(* Logix 5000 project; controller cal1632 1756-L62 rev 16.20; software revision 16.05; part 52 of 61 *)
(* tags used below, declared in another part *)
   FAULT : BOOL;
   HMI : BOOL;
   p01_param_turret_dia_ft : REAL;
   p01r09_pb_global_reset : BOOL;
   p02_real_from_hmi : hmi_real;
   p29_ai_wa_amps : REAL;
   p29_ai_wa_dia_ft : REAL;
   p29_ai_wa_speed : REAL;
   p29_ai_wa_torque : REAL;
   p29_ai_wb_amps : REAL;
   p29_ai_wb_dia_ft : REAL;
   p29_ai_wb_speed : REAL;
   p29_ai_wb_torque : REAL;
   p29_ai_wdr_dia_in : REAL;
   p29_ai_wdr_lc : REAL;
   p29_ai_wdr_turret_amps : REAL;
   p29_ai_wdr_turret_hz : REAL;
   p29_ai_wdr_turret_speed : REAL;
   p29_ao_wda_vfd : REAL;
   p29_ao_wdb_vfd : REAL;
   p29_ao_wdr_turret_selected_speed : REAL;
   p29_ao_wdra_selected_speed : REAL;
   p29_ao_wdrb_selected_speed : REAL;
   p29_di_wdr_turret : acs800_di_normal;
   p29_dint_to_hmi : DINT[16];
   p29_do_wdr_turret : acs800_do_normal;
   p29_param_wa_gear_ratio : REAL;
   p29_param_wb_gear_ratio : REAL;
   p29_param_wdt_gear_ratio : REAL;
   p29_real_to_hmi : REAL[112];
   p29_wda_control_word : INT;
   p29_wda_status_word : INT;
   p29_wda_vfd_input_max : REAL;
   p29_wda_vfd_input_min : REAL;
   p29_wda_vfd_output_max : REAL;
   p29_wda_vfd_output_min : REAL;
   p29_wdb_control_word : INT;
   p29_wdb_status_word : INT;
   p29_wdb_vfd_input_max : REAL;
   p29_wdb_vfd_input_min : REAL;
   p29_wdb_vfd_output_max : REAL;
   p29_wdb_vfd_output_min : REAL;
   p29r01 : routine;
   p29r03_wa_tq_fifo : CONTROL;
   p29r04 : routine;
   p29r04_timer_fault : TIMER[4];
   p29r04_timer_warning : TIMER[4];
   p29r04_wda_vfd_out_scaling : SYS_SCP;
   p29r04_wdb_vfd_out_scaling : SYS_SCP;
   p29r04_wdr_turret_speed_to_vfd : SYS_SPEED_TO_VFD;
   p29r04_wdra_speed_to_vfd : SYS_SPEED_TO_VFD;
   p29r04_wdrb_speed_to_vfd : SYS_SPEED_TO_VFD;
   p29r05 : routine;
   p29r05_timer_fault : TIMER[4];
   p29r05_timer_warning : TIMER[4];
   p29r06 : routine;
   p29r06_ave_wdr_lc : REAL;
   p29r06_lc_buffer : REAL[20];
   p29r06_sample_timer : TIMER;
   p29r06_timer_fault : TIMER[4];
   p29r06_timer_warning : TIMER[4];
   p29r06_unload : REAL;
   p29r06_wdr_lc_ave_ctrl : CONTROL;
   p29r06_wdr_lc_fifo : CONTROL;
   p29r13_ai_wa_footage_ft : REAL;
   p29r13_ai_wb_footage_ft : REAL;
   p29r15_ao_torque : REAL;
   p29r15_wdra_active : BOOL;
   p29r16_ao_torque : REAL;
   p29r16_wdrb_active : BOOL;
   p29r17_winder_a_avg_diam_inch : REAL;
   p29r18_winder_b_avg_diam_inch : REAL;
   p29r20_index_complete : BOOL;
   turret_in_position : BOOL;   // Turret In Position
(* P29_Winder, continued *)

ROUTINE R04_Output   (* ladder *)
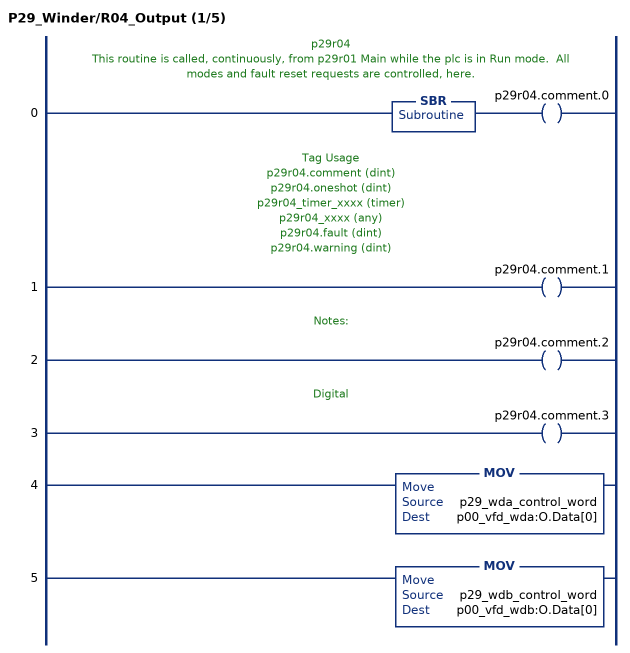
   // p29r04
   // This routine is called, continuously, from p29r01 Main while the plc is in Run mode.  All modes and fault reset requests are controlled, here.
   0: SBR()OTE(p29r04.comment.0);
   // Tag Usage
   // p29r04.comment (dint)
   // p29r04.oneshot (dint)
   // p29r04_timer_xxxx (timer)
   // p29r04_xxxx (any)
   // p29r04.fault (dint)
   // p29r04.warning (dint)
   1: OTE(p29r04.comment.1);
   // Notes:
   2: OTE(p29r04.comment.2);
   // Digital
   3: OTE(p29r04.comment.3);
   4: MOV(p29_wda_control_word,p00_vfd_wda:O.Data[0]);
   5: MOV(p29_wdb_control_word,p00_vfd_wdb:O.Data[0]);
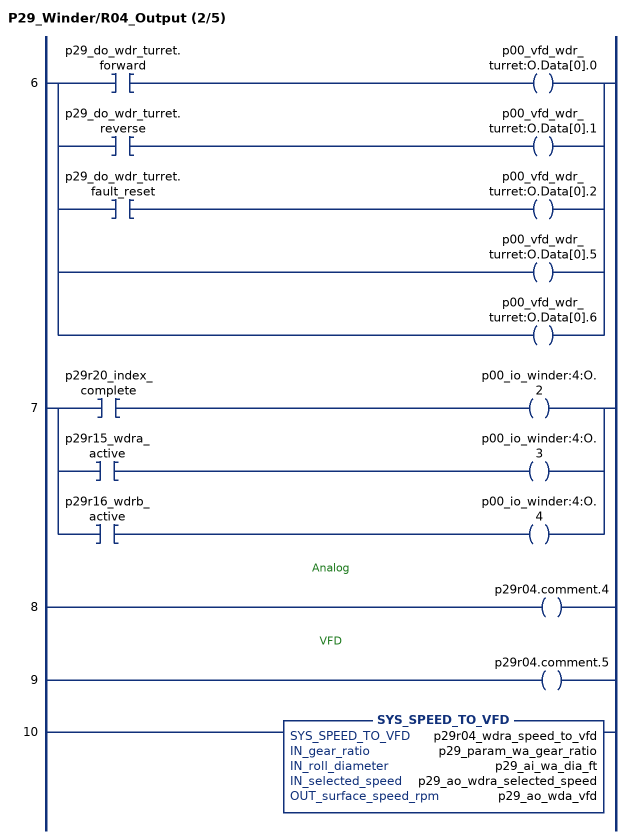
   6: [XIC(p29_do_wdr_turret.forward) OTE(p00_vfd_wdr_turret:O.Data[0].0) ,XIC(p29_do_wdr_turret.reverse) OTE(p00_vfd_wdr_turret:O.Data[0].1) ,XIC(p29_do_wdr_turret.fault_reset) OTE(p00_vfd_wdr_turret:O.Data[0].2) ,OTE(p00_vfd_wdr_turret:O.Data[0].5) ,OTE(p00_vfd_wdr_turret:O.Data[0].6) ];
   7: [XIC(p29r20_index_complete) OTE(p00_io_winder:4:O.2) ,XIC(p29r15_wdra_active) OTE(p00_io_winder:4:O.3) ,XIC(p29r16_wdrb_active) OTE(p00_io_winder:4:O.4) ];
   // Analog
   8: OTE(p29r04.comment.4);
   // VFD
   9: OTE(p29r04.comment.5);
   10: SYS_SPEED_TO_VFD(p29r04_wdra_speed_to_vfd,p29_param_wa_gear_ratio,p29_ai_wa_dia_ft,p29_ao_wdra_selected_speed,p29_ao_wda_vfd);
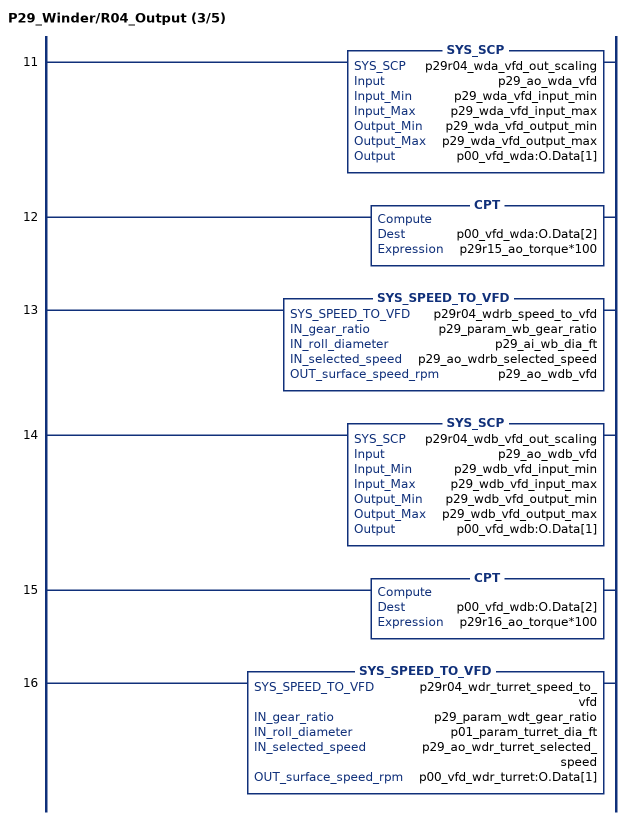
   11: SYS_SCP(p29r04_wda_vfd_out_scaling,p29_ao_wda_vfd,p29_wda_vfd_input_min,p29_wda_vfd_input_max,p29_wda_vfd_output_min,p29_wda_vfd_output_max,p00_vfd_wda:O.Data[1]);
   12: CPT(p00_vfd_wda:O.Data[2],p29r15_ao_torque*100);
   13: SYS_SPEED_TO_VFD(p29r04_wdrb_speed_to_vfd,p29_param_wb_gear_ratio,p29_ai_wb_dia_ft,p29_ao_wdrb_selected_speed,p29_ao_wdb_vfd);
   14: SYS_SCP(p29r04_wdb_vfd_out_scaling,p29_ao_wdb_vfd,p29_wdb_vfd_input_min,p29_wdb_vfd_input_max,p29_wdb_vfd_output_min,p29_wdb_vfd_output_max,p00_vfd_wdb:O.Data[1]);
   15: CPT(p00_vfd_wdb:O.Data[2],p29r16_ao_torque*100);
   16: SYS_SPEED_TO_VFD(p29r04_wdr_turret_speed_to_vfd,p29_param_wdt_gear_ratio,p01_param_turret_dia_ft,p29_ao_wdr_turret_selected_speed,p00_vfd_wdr_turret:O.Data[1]);
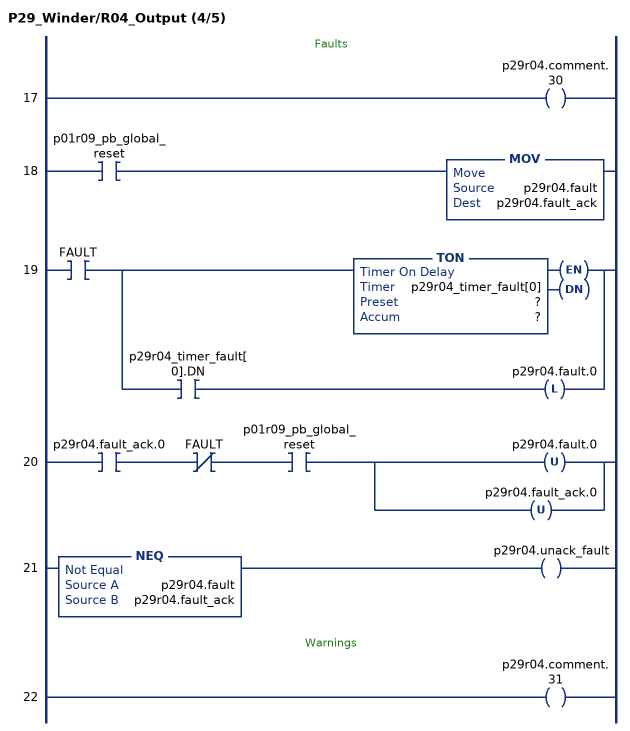
   // Faults
   17: OTE(p29r04.comment.30);
   18: XIC(p01r09_pb_global_reset)MOV(p29r04.fault,p29r04.fault_ack);
   19: XIC(FAULT)[TON(p29r04_timer_fault[0],?,?) ,XIC(p29r04_timer_fault[0].DN) OTL(p29r04.fault.0) ];
   20: XIC(p29r04.fault_ack.0)XIO(FAULT)XIC(p01r09_pb_global_reset)[OTU(p29r04.fault.0) ,OTU(p29r04.fault_ack.0) ];
   21: NEQ(p29r04.fault,p29r04.fault_ack)OTE(p29r04.unack_fault);
   // Warnings
   22: OTE(p29r04.comment.31);
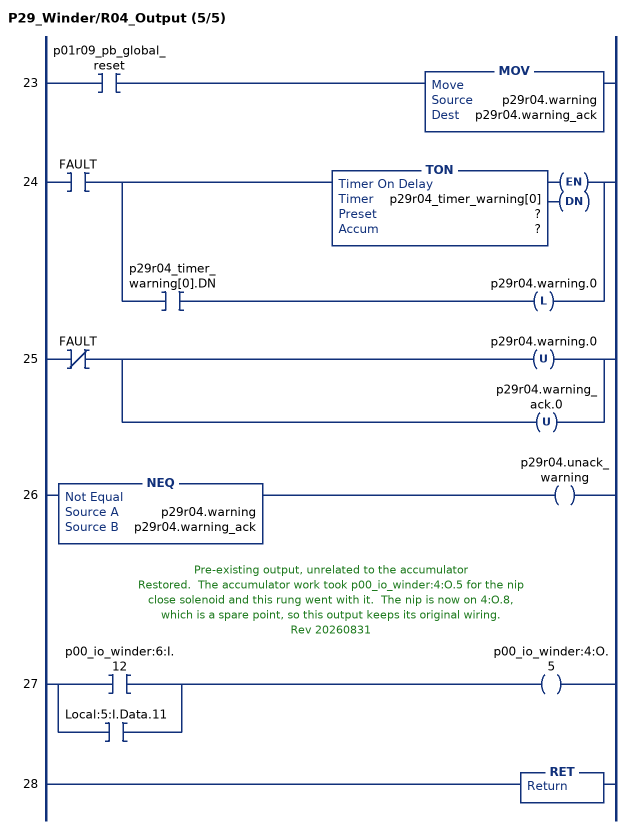
   23: XIC(p01r09_pb_global_reset)MOV(p29r04.warning,p29r04.warning_ack);
   24: XIC(FAULT)[TON(p29r04_timer_warning[0],?,?) ,XIC(p29r04_timer_warning[0].DN) OTL(p29r04.warning.0) ];
   25: XIO(FAULT)[OTU(p29r04.warning.0) ,OTU(p29r04.warning_ack.0) ];
   26: NEQ(p29r04.warning,p29r04.warning_ack)OTE(p29r04.unack_warning);
   // Pre-existing output, unrelated to the accumulator
   // Restored.  The accumulator work took p00_io_winder:4:O.5 for the nip
   // close solenoid and this rung went with it.  The nip is now on 4:O.8,
   // which is a spare point, so this output keeps its original wiring.
   // Rev 20260831
   27: [XIC(p00_io_winder:6:I.12) ,XIC(Local:5:I.Data.11) ]OTE(p00_io_winder:4:O.5);
   28: RET();
END_ROUTINE

ROUTINE R05_Dint_to_HMI   (* ladder *)
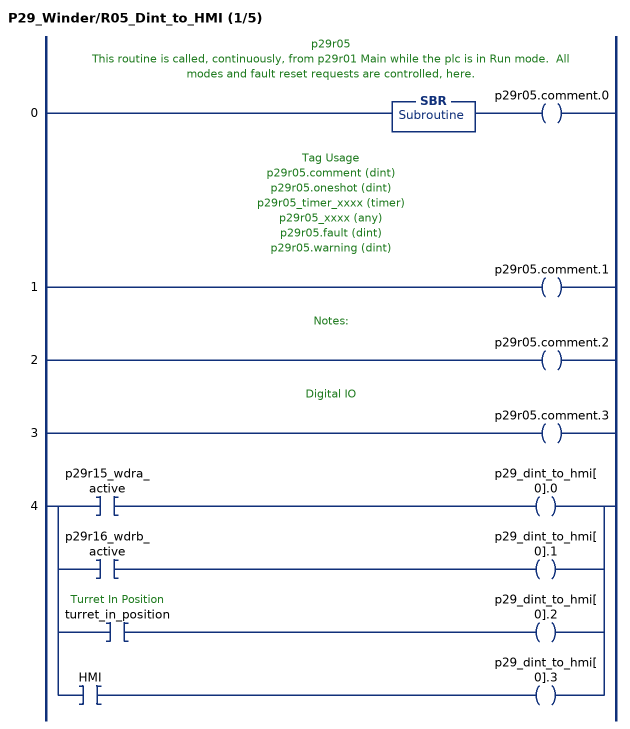
   // p29r05
   // This routine is called, continuously, from p29r01 Main while the plc is in Run mode.  All modes and fault reset requests are controlled, here.
   0: SBR()OTE(p29r05.comment.0);
   // Tag Usage
   // p29r05.comment (dint)
   // p29r05.oneshot (dint)
   // p29r05_timer_xxxx (timer)
   // p29r05_xxxx (any)
   // p29r05.fault (dint)
   // p29r05.warning (dint)
   1: OTE(p29r05.comment.1);
   // Notes:
   2: OTE(p29r05.comment.2);
   // Digital IO
   3: OTE(p29r05.comment.3);
   4: [XIC(p29r15_wdra_active) OTE(p29_dint_to_hmi[0].0) ,XIC(p29r16_wdrb_active) OTE(p29_dint_to_hmi[0].1) ,XIC(turret_in_position) OTE(p29_dint_to_hmi[0].2) ,XIC(HMI) OTE(p29_dint_to_hmi[0].3) ];
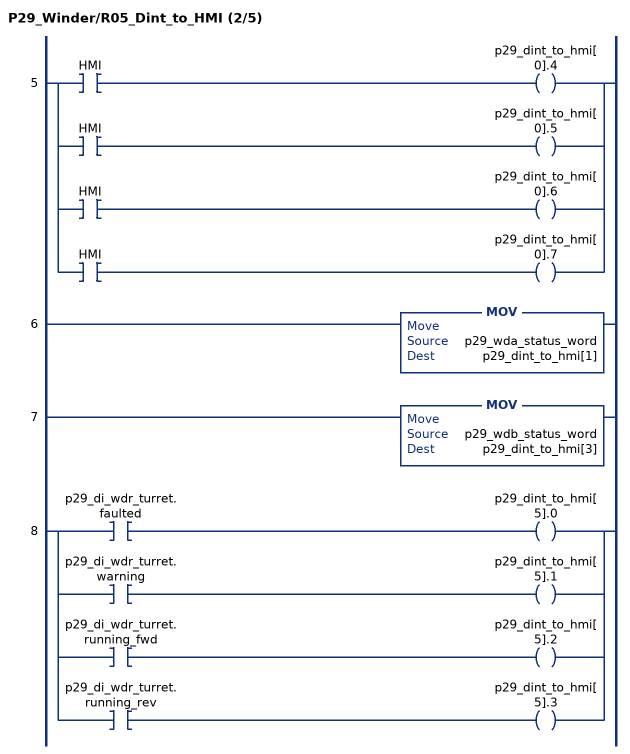
   5: [XIC(HMI) OTE(p29_dint_to_hmi[0].4) ,XIC(HMI) OTE(p29_dint_to_hmi[0].5) ,XIC(HMI) OTE(p29_dint_to_hmi[0].6) ,XIC(HMI) OTE(p29_dint_to_hmi[0].7) ];
   6: MOV(p29_wda_status_word,p29_dint_to_hmi[1]);
   7: MOV(p29_wdb_status_word,p29_dint_to_hmi[3]);
   8: [XIC(p29_di_wdr_turret.faulted) OTE(p29_dint_to_hmi[5].0) ,XIC(p29_di_wdr_turret.warning) OTE(p29_dint_to_hmi[5].1) ,XIC(p29_di_wdr_turret.running_fwd) OTE(p29_dint_to_hmi[5].2) ,XIC(p29_di_wdr_turret.running_rev) OTE(p29_dint_to_hmi[5].3) ];
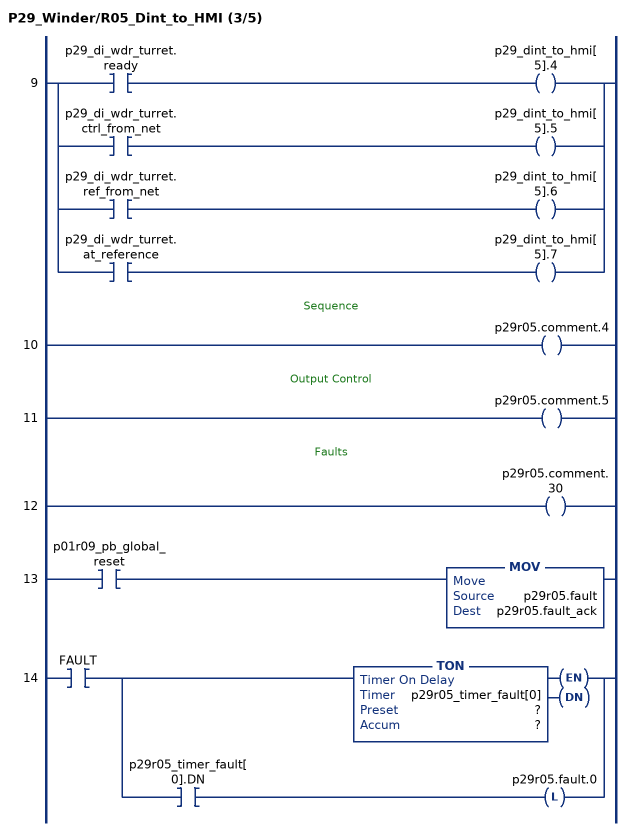
   9: [XIC(p29_di_wdr_turret.ready) OTE(p29_dint_to_hmi[5].4) ,XIC(p29_di_wdr_turret.ctrl_from_net) OTE(p29_dint_to_hmi[5].5) ,XIC(p29_di_wdr_turret.ref_from_net) OTE(p29_dint_to_hmi[5].6) ,XIC(p29_di_wdr_turret.at_reference) OTE(p29_dint_to_hmi[5].7) ];
   // Sequence
   10: OTE(p29r05.comment.4);
   // Output Control
   11: OTE(p29r05.comment.5);
   // Faults
   12: OTE(p29r05.comment.30);
   13: XIC(p01r09_pb_global_reset)MOV(p29r05.fault,p29r05.fault_ack);
   14: XIC(FAULT)[TON(p29r05_timer_fault[0],?,?) ,XIC(p29r05_timer_fault[0].DN) OTL(p29r05.fault.0) ];
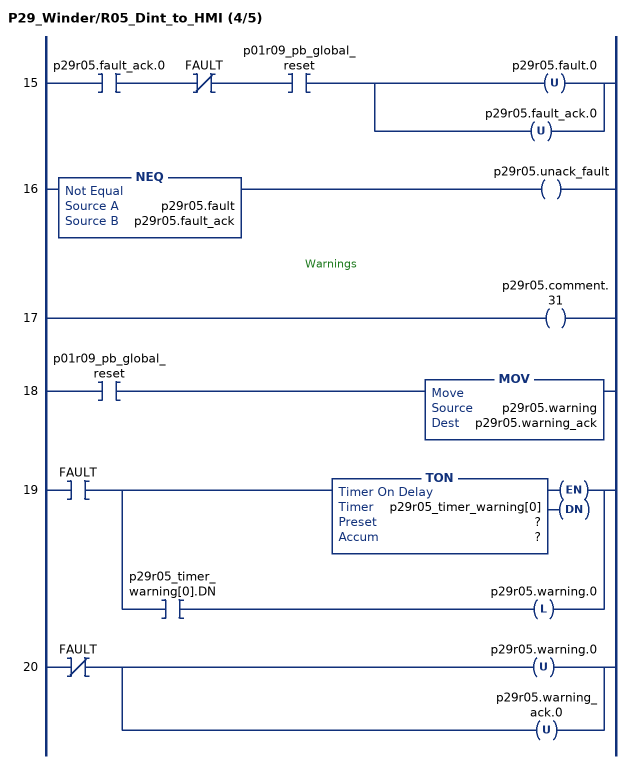
   15: XIC(p29r05.fault_ack.0)XIO(FAULT)XIC(p01r09_pb_global_reset)[OTU(p29r05.fault.0) ,OTU(p29r05.fault_ack.0) ];
   16: NEQ(p29r05.fault,p29r05.fault_ack)OTE(p29r05.unack_fault);
   // Warnings
   17: OTE(p29r05.comment.31);
   18: XIC(p01r09_pb_global_reset)MOV(p29r05.warning,p29r05.warning_ack);
   19: XIC(FAULT)[TON(p29r05_timer_warning[0],?,?) ,XIC(p29r05_timer_warning[0].DN) OTL(p29r05.warning.0) ];
   20: XIO(FAULT)[OTU(p29r05.warning.0) ,OTU(p29r05.warning_ack.0) ];
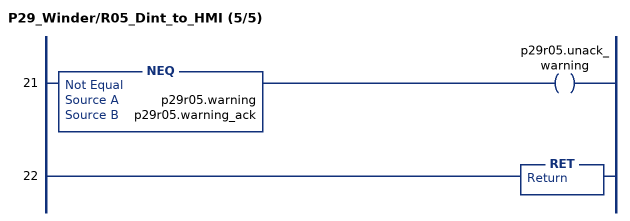
   21: NEQ(p29r05.warning,p29r05.warning_ack)OTE(p29r05.unack_warning);
   22: RET();
END_ROUTINE

ROUTINE R06_Real_to_HMI   (* ladder *)
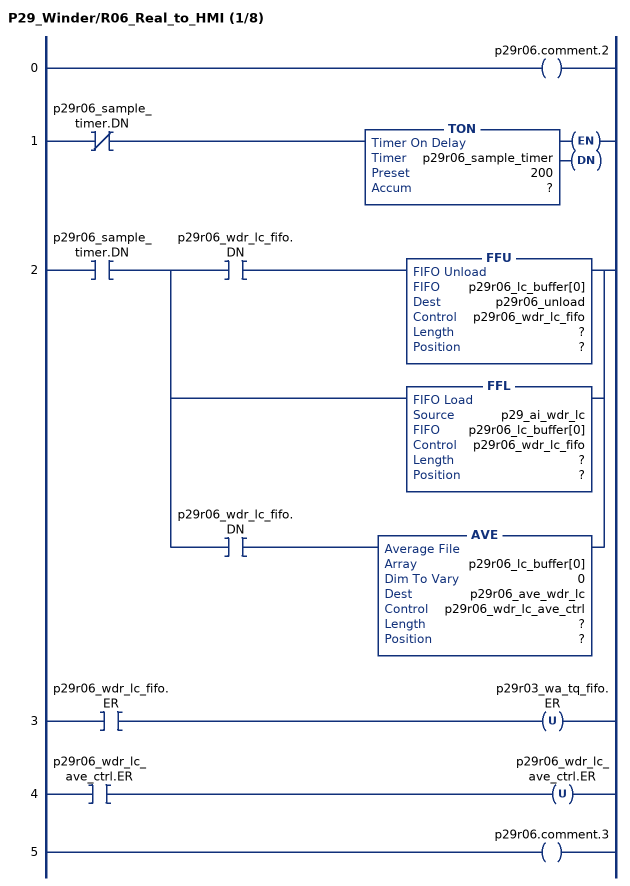
   0: OTE(p29r06.comment.2);
   1: XIO(p29r06_sample_timer.DN)TON(p29r06_sample_timer,?,?);
   2: XIC(p29r06_sample_timer.DN)[XIC(p29r06_wdr_lc_fifo.DN) FFU(p29r06_lc_buffer[0],p29r06_unload,p29r06_wdr_lc_fifo,?,?) ,FFL(p29_ai_wdr_lc,p29r06_lc_buffer[0],p29r06_wdr_lc_fifo,?,?) ,XIC(p29r06_wdr_lc_fifo.DN) AVE(p29r06_lc_buffer[0],0,p29r06_ave_wdr_lc,p29r06_wdr_lc_ave_ctrl,?,?) ];
   3: XIC(p29r06_wdr_lc_fifo.ER)OTU(p29r03_wa_tq_fifo.ER);
   4: XIC(p29r06_wdr_lc_ave_ctrl.ER)OTU(p29r06_wdr_lc_ave_ctrl.ER);
   5: OTE(p29r06.comment.3);
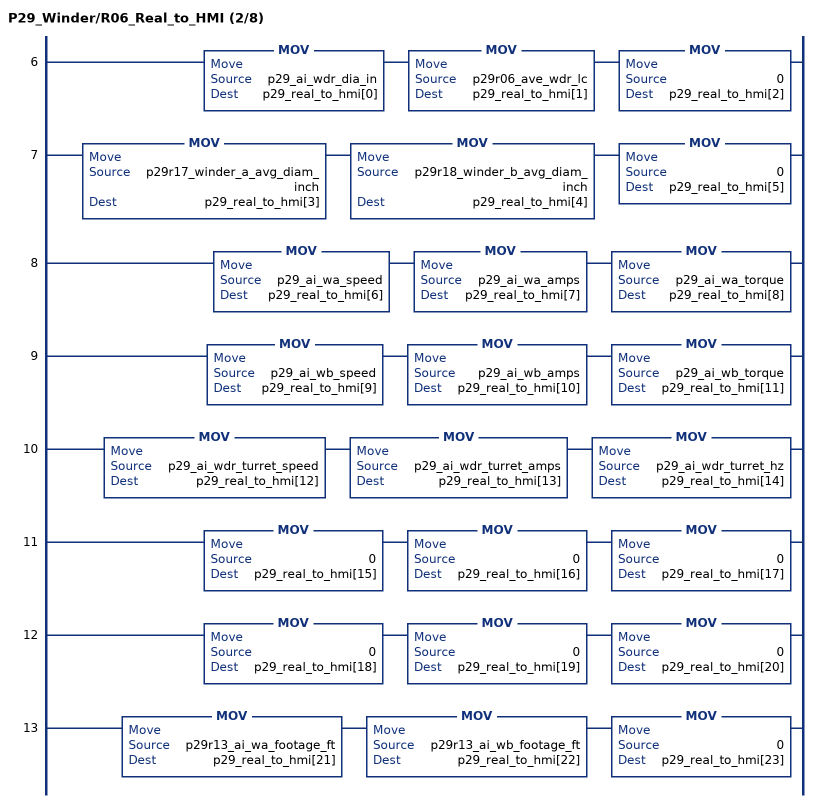
   6: MOV(p29_ai_wdr_dia_in,p29_real_to_hmi[0])MOV(p29r06_ave_wdr_lc,p29_real_to_hmi[1])MOV(0,p29_real_to_hmi[2]);
   7: MOV(p29r17_winder_a_avg_diam_inch,p29_real_to_hmi[3])MOV(p29r18_winder_b_avg_diam_inch,p29_real_to_hmi[4])MOV(0,p29_real_to_hmi[5]);
   8: MOV(p29_ai_wa_speed,p29_real_to_hmi[6])MOV(p29_ai_wa_amps,p29_real_to_hmi[7])MOV(p29_ai_wa_torque,p29_real_to_hmi[8]);
   9: MOV(p29_ai_wb_speed,p29_real_to_hmi[9])MOV(p29_ai_wb_amps,p29_real_to_hmi[10])MOV(p29_ai_wb_torque,p29_real_to_hmi[11]);
   10: MOV(p29_ai_wdr_turret_speed,p29_real_to_hmi[12])MOV(p29_ai_wdr_turret_amps,p29_real_to_hmi[13])MOV(p29_ai_wdr_turret_hz,p29_real_to_hmi[14]);
   11: MOV(0,p29_real_to_hmi[15])MOV(0,p29_real_to_hmi[16])MOV(0,p29_real_to_hmi[17]);
   12: MOV(0,p29_real_to_hmi[18])MOV(0,p29_real_to_hmi[19])MOV(0,p29_real_to_hmi[20]);
   13: MOV(p29r13_ai_wa_footage_ft,p29_real_to_hmi[21])MOV(p29r13_ai_wb_footage_ft,p29_real_to_hmi[22])MOV(0,p29_real_to_hmi[23]);
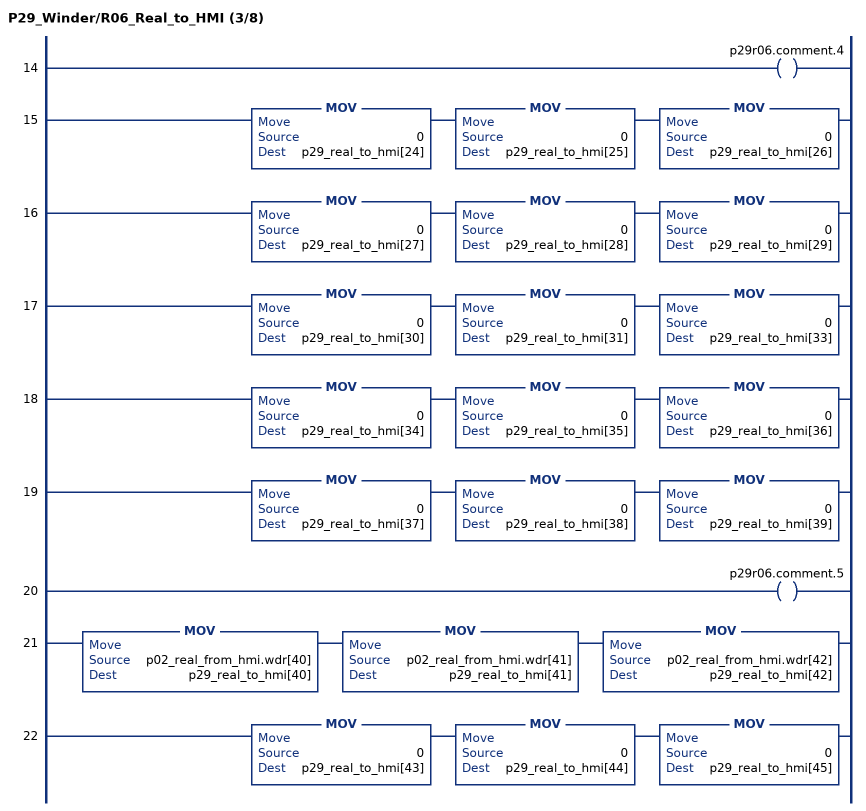
   14: OTE(p29r06.comment.4);
   15: MOV(0,p29_real_to_hmi[24])MOV(0,p29_real_to_hmi[25])MOV(0,p29_real_to_hmi[26]);
   16: MOV(0,p29_real_to_hmi[27])MOV(0,p29_real_to_hmi[28])MOV(0,p29_real_to_hmi[29]);
   17: MOV(0,p29_real_to_hmi[30])MOV(0,p29_real_to_hmi[31])MOV(0,p29_real_to_hmi[33]);
   18: MOV(0,p29_real_to_hmi[34])MOV(0,p29_real_to_hmi[35])MOV(0,p29_real_to_hmi[36]);
   19: MOV(0,p29_real_to_hmi[37])MOV(0,p29_real_to_hmi[38])MOV(0,p29_real_to_hmi[39]);
   20: OTE(p29r06.comment.5);
   21: MOV(p02_real_from_hmi.wdr[40],p29_real_to_hmi[40])MOV(p02_real_from_hmi.wdr[41],p29_real_to_hmi[41])MOV(p02_real_from_hmi.wdr[42],p29_real_to_hmi[42]);
   22: MOV(0,p29_real_to_hmi[43])MOV(0,p29_real_to_hmi[44])MOV(0,p29_real_to_hmi[45]);
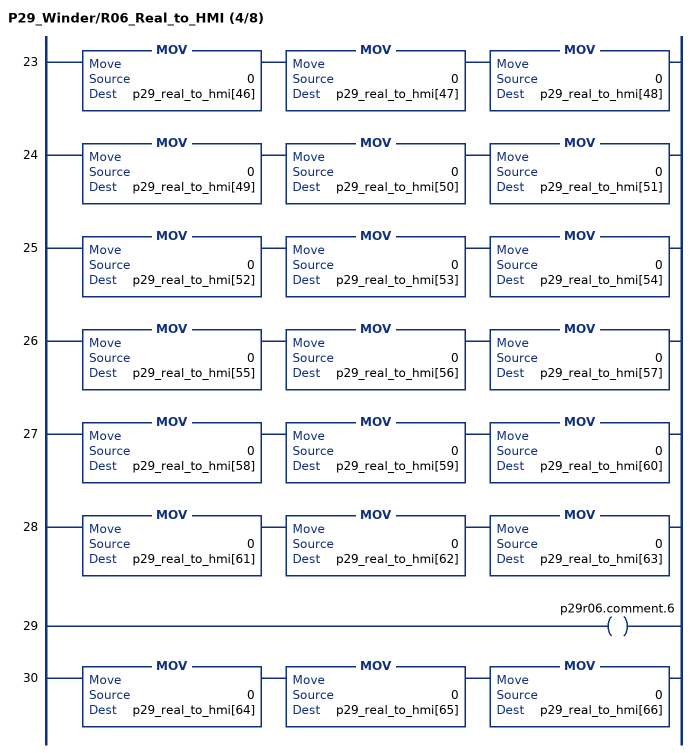
   23: MOV(0,p29_real_to_hmi[46])MOV(0,p29_real_to_hmi[47])MOV(0,p29_real_to_hmi[48]);
   24: MOV(0,p29_real_to_hmi[49])MOV(0,p29_real_to_hmi[50])MOV(0,p29_real_to_hmi[51]);
   25: MOV(0,p29_real_to_hmi[52])MOV(0,p29_real_to_hmi[53])MOV(0,p29_real_to_hmi[54]);
   26: MOV(0,p29_real_to_hmi[55])MOV(0,p29_real_to_hmi[56])MOV(0,p29_real_to_hmi[57]);
   27: MOV(0,p29_real_to_hmi[58])MOV(0,p29_real_to_hmi[59])MOV(0,p29_real_to_hmi[60]);
   28: MOV(0,p29_real_to_hmi[61])MOV(0,p29_real_to_hmi[62])MOV(0,p29_real_to_hmi[63]);
   29: OTE(p29r06.comment.6);
   30: MOV(0,p29_real_to_hmi[64])MOV(0,p29_real_to_hmi[65])MOV(0,p29_real_to_hmi[66]);
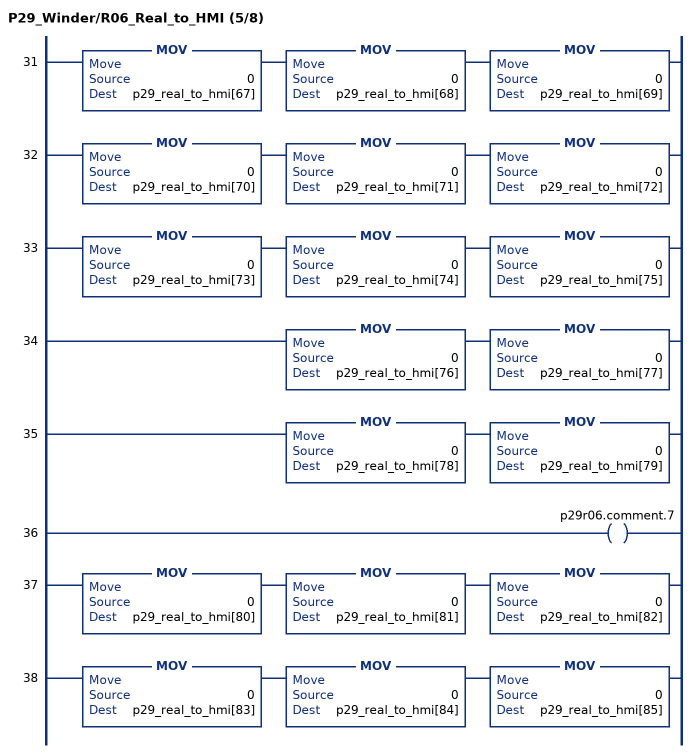
   31: MOV(0,p29_real_to_hmi[67])MOV(0,p29_real_to_hmi[68])MOV(0,p29_real_to_hmi[69]);
   32: MOV(0,p29_real_to_hmi[70])MOV(0,p29_real_to_hmi[71])MOV(0,p29_real_to_hmi[72]);
   33: MOV(0,p29_real_to_hmi[73])MOV(0,p29_real_to_hmi[74])MOV(0,p29_real_to_hmi[75]);
   34: MOV(0,p29_real_to_hmi[76])MOV(0,p29_real_to_hmi[77]);
   35: MOV(0,p29_real_to_hmi[78])MOV(0,p29_real_to_hmi[79]);
   36: OTE(p29r06.comment.7);
   37: MOV(0,p29_real_to_hmi[80])MOV(0,p29_real_to_hmi[81])MOV(0,p29_real_to_hmi[82]);
   38: MOV(0,p29_real_to_hmi[83])MOV(0,p29_real_to_hmi[84])MOV(0,p29_real_to_hmi[85]);
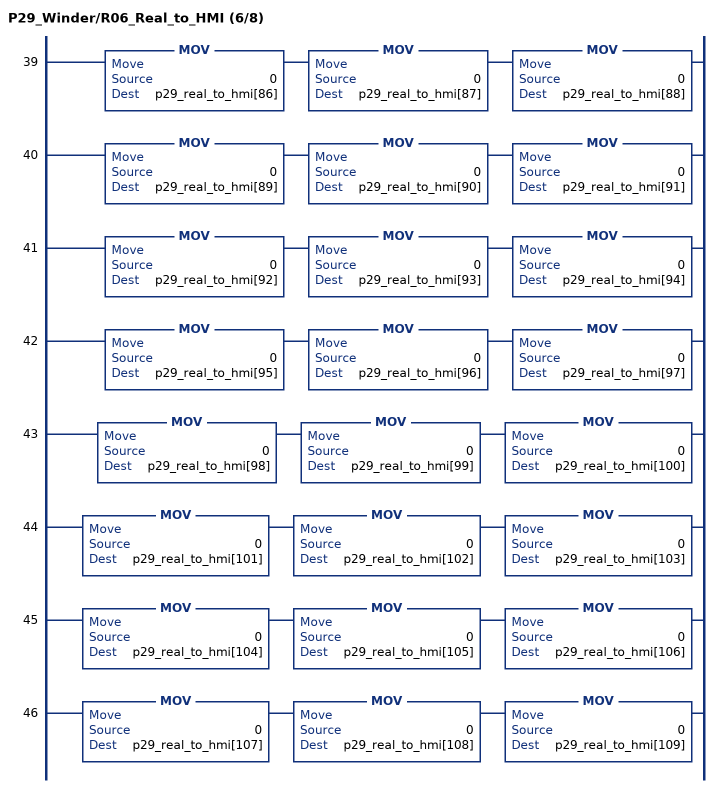
   39: MOV(0,p29_real_to_hmi[86])MOV(0,p29_real_to_hmi[87])MOV(0,p29_real_to_hmi[88]);
   40: MOV(0,p29_real_to_hmi[89])MOV(0,p29_real_to_hmi[90])MOV(0,p29_real_to_hmi[91]);
   41: MOV(0,p29_real_to_hmi[92])MOV(0,p29_real_to_hmi[93])MOV(0,p29_real_to_hmi[94]);
   42: MOV(0,p29_real_to_hmi[95])MOV(0,p29_real_to_hmi[96])MOV(0,p29_real_to_hmi[97]);
   43: MOV(0,p29_real_to_hmi[98])MOV(0,p29_real_to_hmi[99])MOV(0,p29_real_to_hmi[100]);
   44: MOV(0,p29_real_to_hmi[101])MOV(0,p29_real_to_hmi[102])MOV(0,p29_real_to_hmi[103]);
   45: MOV(0,p29_real_to_hmi[104])MOV(0,p29_real_to_hmi[105])MOV(0,p29_real_to_hmi[106]);
   46: MOV(0,p29_real_to_hmi[107])MOV(0,p29_real_to_hmi[108])MOV(0,p29_real_to_hmi[109]);
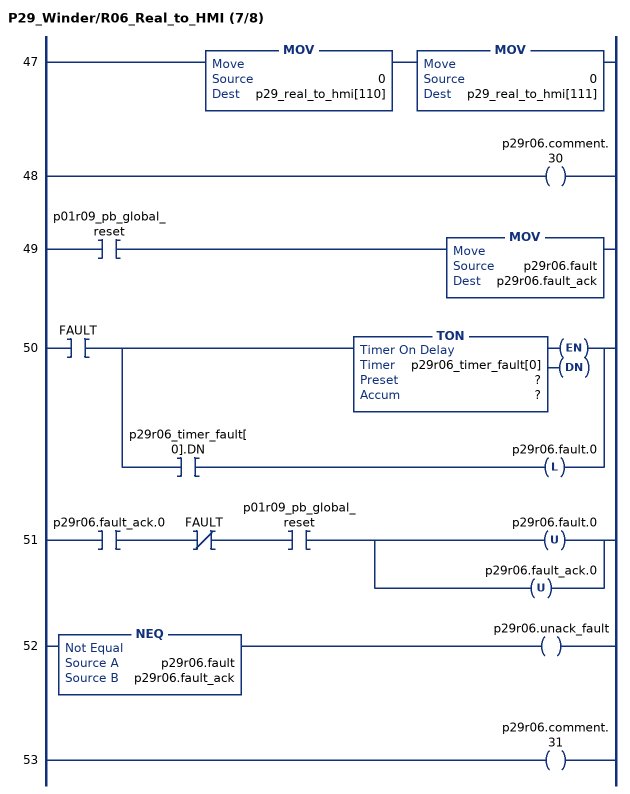
   47: MOV(0,p29_real_to_hmi[110])MOV(0,p29_real_to_hmi[111]);
   48: OTE(p29r06.comment.30);
   49: XIC(p01r09_pb_global_reset)MOV(p29r06.fault,p29r06.fault_ack);
   50: XIC(FAULT)[TON(p29r06_timer_fault[0],?,?) ,XIC(p29r06_timer_fault[0].DN) OTL(p29r06.fault.0) ];
   51: XIC(p29r06.fault_ack.0)XIO(FAULT)XIC(p01r09_pb_global_reset)[OTU(p29r06.fault.0) ,OTU(p29r06.fault_ack.0) ];
   52: NEQ(p29r06.fault,p29r06.fault_ack)OTE(p29r06.unack_fault);
   53: OTE(p29r06.comment.31);
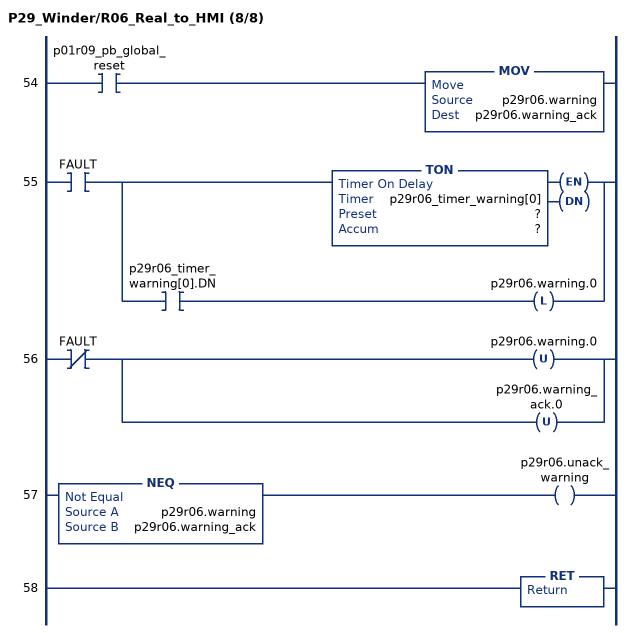
   54: XIC(p01r09_pb_global_reset)MOV(p29r06.warning,p29r06.warning_ack);
   55: XIC(FAULT)[TON(p29r06_timer_warning[0],?,?) ,XIC(p29r06_timer_warning[0].DN) OTL(p29r06.warning.0) ];
   56: XIO(FAULT)[OTU(p29r06.warning.0) ,OTU(p29r06.warning_ack.0) ];
   57: NEQ(p29r06.warning,p29r06.warning_ack)OTE(p29r06.unack_warning);
   58: RET();
END_ROUTINE
